// TIA Portal V18 export
DATA_BLOCK "PC"   // DB69
{ S7_Optimized_Access := 'FALSE'; DB_Accessible_From_OPC_UA := 'FALSE' }
VERSION : 0.1
// stored: AutoNumber false, DBAccessibleFromOPCUA false, IsOnlyStoredInLoadMemory false, IsWriteProtectedInAS false
   VAR
      Keep_alive_fromPLC : Bool;
      X_ray_ready_fromPLC : Bool;
      Image_ready_fromPC : Bool;
      PLC_RESET_Image_ready_fromPC : Bool;
      POS_M1Z : Real;
      POS_M2Y : Real;
      POS_M3X : Real;
      POS_M4O1Tilt : Real;
      POS_M5O2Rot : Real;
   END_VAR
BEGIN
END_DATA_BLOCK
